FUNCTION_BLOCK FB_StaticMatrix_Test EXTENDS FB_TestSuite
VAR_INPUT
END_VAR
VAR_OUTPUT
END_VAR
VAR
END_VAR

WhenCreatedExpectDataAssignable();

METHOD PRIVATE WhenCreatedExpectDataAssignable
VAR_INPUT
END_VAR
VAR
	M1 : ExternalStaticMatrix;
	M2 : DynamicMatrix;
	Data : ARRAY[0..8] OF LREAL;
	
	
END_VAR
TEST('WhenCreatedExpectDataAssignable');

// @TEST-RUN
M2.InitMagicSquare(3);
M1.Init(ADR(Data),3,3);
M1.FillFrom(M2);


// @TEST-ASSERT
AssertTrue(M1.IsEqual(M2),'Data was not all assigned');

TEST_FINISHED();
END_METHOD

END_FUNCTION_BLOCK

(* stored: Version 1.1.0.1, ProductVersion 3.1.4024.9
   POU FB_StaticMatrix_Test: Id {87892744-99b1-0998-358b-247090a4c803}, SpecialFunc None
   Method WhenCreatedExpectDataAssignable: Id {3d9f6a97-0f3a-0add-2595-58c98258ff46} *)
